// TIA Portal V20 export
VAR_GLOBAL   // PLC tag table "Cabinet_1"
   Sz1_St25_SenA AT %I1100.0 : Bool;
   Sz1_St25_SenB AT %I1100.1 : Bool;
   Sz1_St25_SenC AT %I1100.2 : Bool;
   Sz1_St25_SenD AT %I1100.3 : Bool;
   Sz1_St26_SenA AT %I1100.4 : Bool;
   Sz1_St26_SenB AT %I1100.5 : Bool;
   Sz1_St26_SenC AT %I1100.6 : Bool;
   Sz1_St26_SenD AT %I1100.7 : Bool;
   Sz1_St23_SenA AT %I1101.0 : Bool;
   Sz1_St23_SenB AT %I1101.1 : Bool;
   Sz1_St23_SenC AT %I1101.2 : Bool;
   Sz1_St23_SenD AT %I1101.3 : Bool;
   Sz1_St24_SenA AT %I1101.4 : Bool;
   Sz1_St24_SenB AT %I1101.5 : Bool;
   Sz1_St24_SenC AT %I1101.6 : Bool;
   Sz1_St24_SenD AT %I1101.7 : Bool;
   Sz1_Button_ST25_ST26 AT %I1102.0 : Bool;
   Sz1_Button_ST26_ST27 AT %I1102.1 : Bool;
   Sz1_Button_ST24_ST23 AT %I1102.2 : Bool;
   Sz1_Button_ST23_ST22 AT %I1102.3 : Bool;
   Sz1_Button_ST24_Seq_Backward AT %I1102.4 : Bool;
   Sz1_Button_ST24_Seq_Forward AT %I1102.5 : Bool;
   Sz1_Button_ST25_Seq_Backward AT %I1102.6 : Bool;
   Sz1_Button_ST25_Seq_Forward AT %I1102.7 : Bool;
   Sz1_Button_ST23_Seq_Forward AT %I1103.0 : Bool;
   Sz1_Button_SS_Down AT %I1103.1 : Bool;
   Sz1_Button_SS_Up AT %I1103.2 : Bool;
   Sz1_Button_SS_Drive_ST25 AT %I1103.3 : Bool;
   Sz1_Button_SS_Drive_ST24 AT %I1103.4 : Bool;
   Sz1_Button_SS_Drive_ST17 AT %I1103.5 : Bool;
   Sz1_Button_SS_Drive_ST14 AT %I1103.6 : Bool;
   "Reserved(1)" AT %I1103.7 : Bool;
   Sz1_Safety1_1 AT %I1150.0 : Bool;
   Sz13_Safety1_1 AT %I1150.1 : Bool;
   "Reserved(12)" AT %I1150.2 : Bool;
   "Reserved(13)" AT %I1150.3 : Bool;
   Sz1_Safety1_2 AT %I1150.4 : Bool;
   Sz13_Safety1_2 AT %I1150.5 : Bool;
   "Reserved(15)" AT %I1150.6 : Bool;
   "Reserved(16)" AT %I1150.7 : Bool;
   "Reserved(17)" AT %I1151.0 : Bool;
   "Reserved(18)" AT %I1151.1 : Bool;
   "Reserved(19)" AT %I1151.2 : Bool;
   "Reserved(20)" AT %I1151.3 : Bool;
   "Reserved(21)" AT %I1151.4 : Bool;
   "Reserved(22)" AT %I1151.5 : Bool;
   "Reserved(23)" AT %I1151.6 : Bool;
   "Reserved(24)" AT %I1151.7 : Bool;
   Sz1_Button_LED_ST25_ST26 AT %Q1100.0 : Bool;
   Sz1_Button_LED_ST26_ST27 AT %Q1100.1 : Bool;
   Sz1_Button_LED_ST24_ST23 AT %Q1100.2 : Bool;
   Sz1_Button_LED_ST23_ST22 AT %Q1100.3 : Bool;
   Sz1_Button_LED_Hyd_Up AT %Q1100.4 : Bool;
   Sz1_Button_LED_Hyd_Down AT %Q1100.5 : Bool;
   Sz1_Button_LED_Air_Up AT %Q1100.6 : Bool;
   Sz1_Button_LED_Air_Down AT %Q1100.7 : Bool;
   Sz1_Button_LED_Wibration AT %Q1101.0 : Bool;
   Sz1_Button_LED_SS_Down AT %Q1101.1 : Bool;
   Sz1_Button_LED_SS_Up AT %Q1101.2 : Bool;
   Sz1_Button_LED_SS_Drive_ST25 AT %Q1101.3 : Bool;
   Sz1_Button_LED_SS_Drive_ST24 AT %Q1101.4 : Bool;
   Sz1_Button_LED_SS_Drive_ST17 AT %Q1101.5 : Bool;
   Sz1_Button_LED_SS_Drive_ST14 AT %Q1101.6 : Bool;
   Reserved AT %Q1101.7 : Bool;
   Sz1_Button_LED_Centering_ST23 AT %Q1102.0 : Bool;
   Sz1_Button_LED_Centering_ST22 AT %Q1102.1 : Bool;
   "Reserved(5)" AT %Q1102.2 : Bool;
   "Reserved(6)" AT %Q1102.3 : Bool;
   Sz1_Button_LED_ST23_Seq_Backward AT %Q1102.4 : Bool;
   ST23_CNT_UPP AT %Q1102.5 : Bool;
   ST23_CNT_V1 AT %Q1102.6 : Bool;
   ST23_CNT_V2 AT %Q1102.7 : Bool;
   iSR_Distance_Value AT %IW502 : Int;
   Sz1_Button_ST23_Seq_Backward AT %I1124.0 : Bool;
   "reserved(2)" AT %I1124.1 : Bool;
   "reserved(3)" AT %I1124.2 : Bool;
   Sz1_Button_Centering_ST23 AT %I1124.3 : Bool;
   Sz1_Button_Centering_ST22 AT %I1124.4 : Bool;
   Reserved_1 AT %I1124.5 : Bool;
   Reserved_2 AT %I1124.6 : Bool;
   Reserved_3 AT %I1124.7 : Bool;
   Reserved_4 AT %I1125.0 : Bool;
   Reserved_5 AT %I1125.1 : Bool;
   Reserved_6 AT %I1125.2 : Bool;
   Reserved_7 AT %I1125.3 : Bool;
   St23_Centering_Up_2 AT %I1125.4 : Bool;
   St23_Centering_Down_2 AT %I1125.5 : Bool;
   St23_Centering_Down_1 AT %I1125.6 : Bool;
   St23_Centering_Up_1 AT %I1125.7 : Bool;
END_VAR
